// TIA Portal V16 export
// export: Created 2023-01-04T15:44:08.8031791Z, ExportSetting WithDefaults, DisplayName Totally Integrated Automation Portal, DisplayVersion V16, DisplayName TIA Portal Version Control Interface, DisplayVersion V16, DisplayName TIA Portal Openness, DisplayVersion V16, DisplayName STEP 7 Professional, DisplayVersion V16, DisplayName STEP 7 Safety, DisplayVersion V16, DisplayName WinCC Advanced, DisplayVersion V16
FUNCTION_BLOCK "Alarm_Logic"   // FB3, LAD
{ S7_Optimized_Access := 'TRUE' }
VERSION : 0.1
// stored: AutoNumber true, IsIECCheckEnabled false, IsRetainMemResEnabled false, MemoryReserve 100, SetENOAutomatically false, UDAEnableTagReadback false
   VAR_TEMP   // added for the SCL form of the ladder/FBD networks
      _w1 : Bool;
      _w2 : Bool;
      _w3 : Bool;
      _w4 : Bool;
      _w5 : Bool;
      _w6 : Bool;
   END_VAR
BEGIN

REGION Network 1: Bottle Overfilled Alarm
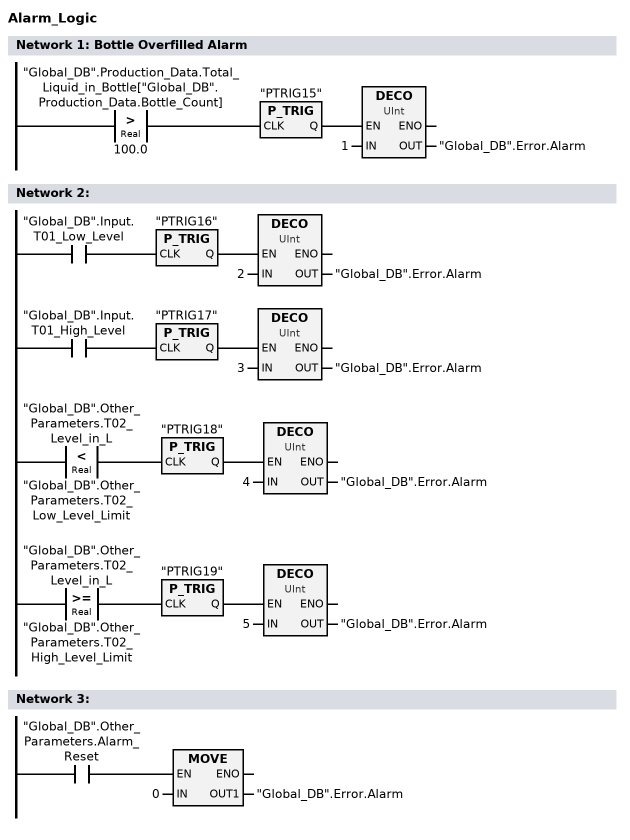
   RUNG wire#powerrail
      { S7_Templates := "SrcType := Real" } GT_Contact(in1 := "Global_DB".Production_Data.Total_Liquid_in_Bottle["Global_DB".Production_Data.Bottle_Count], in2 := 100.0)
      P_Trig( "PTRIG15" )
      { S7_Templates := "[value_type := UInt, return_type := Word]" } DECO(IN := 1, OUT => "Global_DB".Error.Alarm)
   END_RUNG
   // the same network as SCL:
   #_w1 := "Global_DB".Production_Data.Total_Liquid_in_Bottle["Global_DB".Production_Data.Bottle_Count] > 100.0;
   #_w2 := #_w1 AND NOT "PTRIG15";   // rising edge
   "PTRIG15" := #_w1;
   IF #_w2 THEN DECO(IN := 1, OUT => "Global_DB".Error.Alarm); END_IF;
END_REGION

REGION Network 2
   RUNG wire#powerrail
      Contact( "Global_DB".Input.T01_Low_Level )
      P_Trig( "PTRIG16" )
      { S7_Templates := "[value_type := UInt, return_type := Word]" } DECO(IN := 2, OUT => "Global_DB".Error.Alarm)
   END_RUNG
   RUNG wire#powerrail
      Contact( "Global_DB".Input.T01_High_Level )
      P_Trig( "PTRIG17" )
      { S7_Templates := "[value_type := UInt, return_type := Word]" } DECO(IN := 3, OUT => "Global_DB".Error.Alarm)
   END_RUNG
   RUNG wire#powerrail
      { S7_Templates := "SrcType := Real" } LT_Contact(in1 := "Global_DB".Other_Parameters.T02_Level_in_L, in2 := "Global_DB".Other_Parameters.T02_Low_Level_Limit)
      P_Trig( "PTRIG18" )
      { S7_Templates := "[value_type := UInt, return_type := Word]" } DECO(IN := 4, OUT => "Global_DB".Error.Alarm)
   END_RUNG
   RUNG wire#powerrail
      { S7_Templates := "SrcType := Real" } GE_Contact(in1 := "Global_DB".Other_Parameters.T02_Level_in_L, in2 := "Global_DB".Other_Parameters.T02_High_Level_Limit)
      P_Trig( "PTRIG19" )
      { S7_Templates := "[value_type := UInt, return_type := Word]" } DECO(IN := 5, OUT => "Global_DB".Error.Alarm)
   END_RUNG
   // the same network as SCL:
   #_w1 := "Global_DB".Input.T01_Low_Level AND NOT "PTRIG16";   // rising edge
   "PTRIG16" := "Global_DB".Input.T01_Low_Level;
   IF #_w1 THEN DECO(IN := 2, OUT => "Global_DB".Error.Alarm); END_IF;
   #_w2 := "Global_DB".Input.T01_High_Level AND NOT "PTRIG17";   // rising edge
   "PTRIG17" := "Global_DB".Input.T01_High_Level;
   IF #_w2 THEN DECO(IN := 3, OUT => "Global_DB".Error.Alarm); END_IF;
   #_w3 := "Global_DB".Other_Parameters.T02_Level_in_L < "Global_DB".Other_Parameters.T02_Low_Level_Limit;
   #_w4 := #_w3 AND NOT "PTRIG18";   // rising edge
   "PTRIG18" := #_w3;
   IF #_w4 THEN DECO(IN := 4, OUT => "Global_DB".Error.Alarm); END_IF;
   #_w5 := "Global_DB".Other_Parameters.T02_Level_in_L >= "Global_DB".Other_Parameters.T02_High_Level_Limit;
   #_w6 := #_w5 AND NOT "PTRIG19";   // rising edge
   "PTRIG19" := #_w5;
   IF #_w6 THEN DECO(IN := 5, OUT => "Global_DB".Error.Alarm); END_IF;
END_REGION

REGION Network 3
   RUNG wire#powerrail
      Contact( "Global_DB".Other_Parameters.Alarm_Reset )
      Move(in := 0, out1 => "Global_DB".Error.Alarm)
   END_RUNG
   // the same network as SCL:
   IF "Global_DB".Other_Parameters.Alarm_Reset THEN "Global_DB".Error.Alarm := 0; END_IF;
END_REGION
END_FUNCTION_BLOCK
